SUBAPPLICATION Uebung_075 (* MM710 *)
  (* Standard: 61499-2; Description: Copyright (c) 2023 Meisterschulen am Ostbahnhof This program and the accompanying materials are made available under the terms of the Eclipse Public License 2.0 which is available at https://www.eclipse.org/legal/epl-2.0/ SPDX-License-Identifier: EPL-2.0 *)
  (* Version 1.0, 2023-10-23, Franz Höpfinger, Meisterschulen am Ostbahnhof, initial API and implementation and/or initial documentation *)
  PACKAGE Uebungen;
  IMPORT isobus::pgn::ISO_CAN_NODE::NODE1;
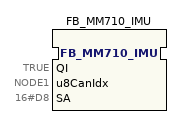
  FBS
    FB_MM710_IMU : logiBUS::bosch::imu::FB_MM710_IMU(QI := TRUE, u8CanIdx := NODE1, SA := 16#D8);
  END_FBS
END_SUBAPPLICATION
